FUNCTION_BLOCK Model_HMI (* Service Interface Function Block Type *)
  (* Standard: 61499-2 *)
  (* Version 0.0, 7/13/2016, Andrei, nxtControl GmbH, template *)
  PACKAGE Main;
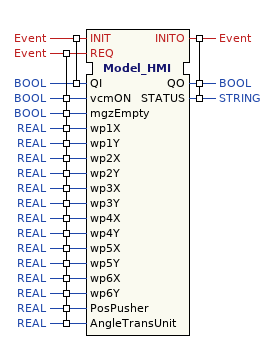
  EVENT_INPUT
    INIT WITH QI;
    REQ WITH vcmON, mgzEmpty, wp1X, wp1Y, wp2X, wp2Y, wp3X, wp3Y, wp4X, wp4Y, wp5X, wp5Y, wp6X, wp6Y, PosPusher, AngleTransUnit;
  END_EVENT
  EVENT_OUTPUT
    INITO WITH QO, STATUS;
  END_EVENT
  VAR_INPUT
    QI : BOOL;
    vcmON : BOOL;
    mgzEmpty : BOOL;
    wp1X : REAL;
    wp1Y : REAL;
    wp2X : REAL;
    wp2Y : REAL;
    wp3X : REAL;
    wp3Y : REAL;
    wp4X : REAL;
    wp4Y : REAL;
    wp5X : REAL;
    wp5Y : REAL;
    wp6X : REAL;
    wp6Y : REAL;
    PosPusher : REAL;
    AngleTransUnit : REAL;
  END_VAR
  VAR_OUTPUT
    QO : BOOL; (* Event Output Qualifier *)
    STATUS : STRING; (* Service Status *)
  END_VAR
  SERVICE /
    SEQUENCE 
    END_SEQUENCE
  END_SERVICE
END_FUNCTION_BLOCK
